KUKA KRL program: chk_w8_wechs_ok.src

&ACCESS RVO12
&COMMENT Check Tool Change
DEF chk_w8_wechs_ok( )

; VERIFICAÇÃO DE FERRAMENTA: TOOL CHANGE

wait for (($in[161]) and ($in[169]) and ($in[177]) and ($in[185]) and (not $in[219]))

END
